FUNCTION_BLOCK Manual_Right
VAR_INPUT
	Input1:BOOL;
	ManualCotrolSpeed	:	REAL;
END_VAR
VAR_OUTPUT
	Flag1:BOOL;
END_VAR
VAR
	temp1:MC_MoveVelocity;
	AxisStop:MC_Stop;
	trig1: F_TRIG;
END_VAR
VAR // added by the converter: edge detectors and wires of the graphical bodies
    _w1 : ANY;
END_VAR

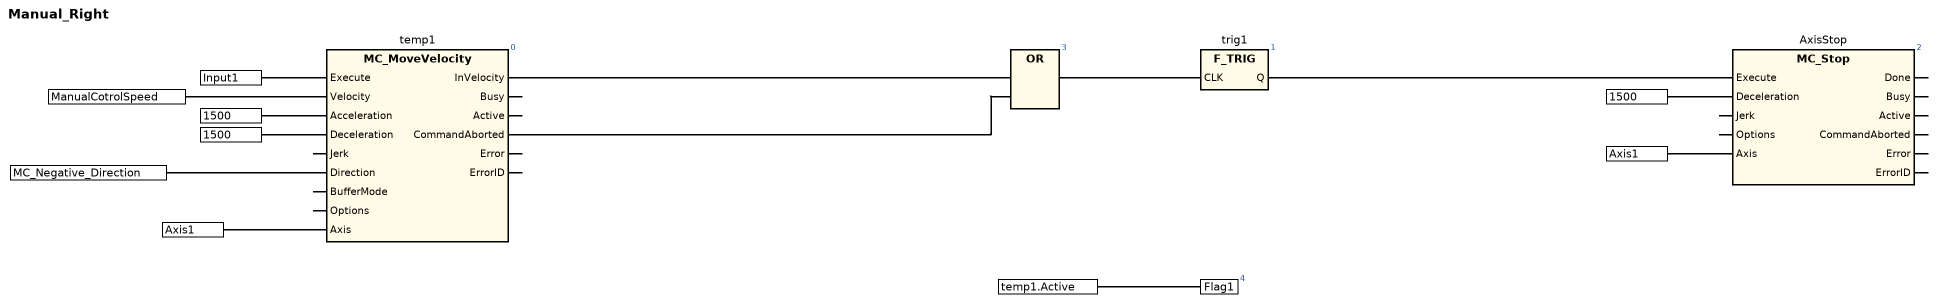
temp1(
    Execute := Input1,
    Velocity := ManualCotrolSpeed,
    Acceleration := 1500,
    Deceleration := 1500,
    Direction := MC_Negative_Direction,
    Axis := Axis1); // MC_MoveVelocity
trig1(CLK := _w1); // F_TRIG
AxisStop(Execute := trig1.Q, Deceleration := 1500, Axis := Axis1); // MC_Stop
_w1 := temp1.InVelocity OR temp1.CommandAborted;
Flag1 := temp1.Active;

END_FUNCTION_BLOCK

(* stored: Version 1.1.0.1, ProductVersion 3.1.4024.12
   POU Manual_Right: Id {b9196604-4d2d-4021-b171-0a8f663713d7}, SpecialFunc None *)
